{attribute 'GeneratedUsingTerminal: BK1250-0000-0000'}
{attribute addProperty BoxType "BK1250-0000-0000"}
{attribute addProperty Id "AdsAddrAT %I*AMSADDR8AoeNetIdAT %I*AMSNETID6StateAT %I*UINT2"}
{attribute addProperty CRC "2417512204"}
{attribute addProperty Size "16"}
TYPE InfoData_90184F0C :
STRUCT
	{attribute addProperty Name "AdsAddr"}
	AdsAddr AT %I* : AMSADDR;
	{attribute addProperty Name "AoeNetId"}
	AoeNetId AT %I* : AMSNETID;
	{attribute addProperty Name "State"}
	State AT %I* : UINT;
END_STRUCT
END_TYPE

(* stored: Version 1.2.0.0, ProductVersion 3.1.4024.9
   DUT InfoData_90184F0C: Id {a0cbd70d-98fc-4099-b8fc-594cb2730c38} *)
